FUNCTION_BLOCK ABSTRACT Motor

METHOD PUBLIC ABSTRACT LoadFuel
END_METHOD

METHOD PUBLIC ABSTRACT SpeedUp
END_METHOD

METHOD PUBLIC ABSTRACT StartUp
END_METHOD

METHOD PUBLIC ABSTRACT Stop
END_METHOD

END_FUNCTION_BLOCK

(* stored: Version 1.1.0.1, ProductVersion 3.1.4024.12
   POU Motor: Id {3f55ef3a-1b19-4ac3-af6a-07651b20dd1a}, SpecialFunc None
   Method LoadFuel: Id {b9f76f1f-c6b9-4a8f-b7ae-3a7493403678}
   Method SpeedUp: Id {76cae08d-6f11-497d-977a-75be8b98cbec}
   Method StartUp: Id {51fbf7ae-0425-47d7-9b55-ca25c5d2db59}
   Method Stop: Id {0af60e0e-884c-449d-b617-42909576f1dc} *)
